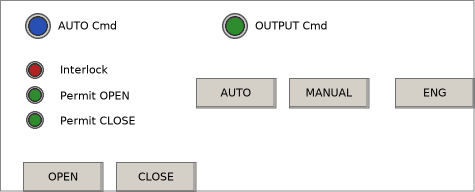
VISUALIZATION GUI_TEMPLATE_ACTUATOR_CMD  // 475x192
VAR_IN_OUT
	m_Instance:	FB_CRYO_ACTUATOR_CMD;
END_VAR
    Lamp1 (25,60 20x20), variable: m_Instance.in_bInterlock, style: Lamp-Lamp1-Red
    Lamp1 (25,85 20x20), variable: m_Instance.bPermitOn, style: Lamp-Lamp1-Green
    Lamp1 (25,110 20x20), variable: m_Instance.bPermitOff, style: Lamp-Lamp1-Green
    Rectangle (57,55 83x30), "Interlock"
    Rectangle (57,81 83x30), "Permit OPEN"
    Rectangle (57,106 83x30), "Permit CLOSE"
    Button (23,162 80x30), "OPEN", colour toggle: (m_Instance.bPermitOn AND NOT m_Instance.bAutoMode) OR m_Instance.bEngMode, input disabled if: m_Instance.bDisableBtnOn
        OnMouseClick: execute { m_Instance.bManualCmd := TRUE; m_Instance.bManualExecute := TRUE; }
    Lamp1 (220,11 30x30), variable: m_Instance.out_Enable, style: Lamp-Lamp1-Green
    Rectangle (252,11 83x30), "OUTPUT Cmd"
    Button (196,78 80x30), "AUTO", colour toggle: m_Instance.bAutoMode, input disabled if: m_Instance.bAutoMode OR m_Instance.bEngMode
        OnMouseClick: execute { m_Instance.bAutoMode := TRUE; }
    Button (289,78 80x30), "MANUAL", colour toggle: NOT m_Instance.bAutoMode, input disabled if: NOT m_Instance.bAutoMode AND NOT_IDLE m_Instance.bEngMode
        OnMouseClick: execute { m_Instance.bAutoMode := FALSE; }
    Button (116,162 80x30), "CLOSE", colour toggle: (m_Instance.bPermitOff AND NOT m_Instance.bAutoMode) OR m_Instance.bEngMode, input disabled if: m_Instance.bDisableBtnOff
        OnMouseClick: execute { m_Instance.bManualCmd := FALSE; m_Instance.bManualExecute := TRUE; }
    Button (395,78 80x30), "ENG", tooltip "Engineering / Commissioning Mode", colour toggle: m_Instance.bEngMode, input disabled if: m_Instance.bAutoMode
        toggle m_Instance.bEngMode
    Lamp1 (23,11 30x30), variable: m_Instance.in_bEnable, style: Lamp-Lamp1-Blue
    Rectangle (55,11 83x30), "AUTO Cmd"
END_VISUALIZATION

(* stored: Version 1.1.0.1, ProductVersion 3.1.4024.9
   Visu GUI_TEMPLATE_ACTUATOR_CMD: Id {f10a6d6e-63ed-40f2-ab1c-f46f44fcd7e5} *)
